// TIA Portal project "hardware_cont" (V17)

(* hardware
DEVICE "S7-1500/ET200MP station_1"  S7-1500 station
   slot 0: "Rail_0"  Rack  6ES7 590-1***0-0AA0
   slot 1: "PLC_1"  CPU 1511-1 PN  6ES7 511-1AK02-0AB0  V2.9
      slot 3: "CPU display_1"  6ES7591-1AA00-0AA0
      slot 32768: "PROFINET interface_1"  X1
         slot 32769: "Port_1"  X1 P1
         slot 32770: "Port_2"  X1 P2
      slot 34817: "Virtual CP interface port_1"  Virtual CP interface port  Virtual CP interface port
   slot 2: "DI 16x24VDC / DQ 16x24VDC/0.5A BA_1"  DI 16x24VDC/DQ 16x24VDC/0.5A BA  6ES7 523-1BL00-0AA0  V1.1
   slot 3: "AI 4xU/I/RTD/TC / AQ 2xU/I ST_1"  AI/AQ 4xU/I/RTD/TC / 2xU/I ST  6ES7 534-7QE00-0AB0  V1.0
   slot 4: "CM PtP RS232 BA_1"  CM PtP RS232 BA  6ES7 540-1AD00-0AA0  V1.0
DEVICE "HMI_2"  TP700 Comfort Outdoor
   slot 0: "HMI_2"  TP700 Comfort Outdoor  6AV2 124-0GC13-0AX0  17.0.0.0
   slot 1: "HMI_RT_2"  TP700 Comfort Outdoor  6AV2 124-0GC13-0AX0  17.0.0.0
   slot 5: "HMI_2.IE_CP_1"  PROFINET Interface  17.0.0.0
      slot 1: "PROFINET Interface_1"  PROFINET Interface
         slot 1: "Port_1"  Port
         slot 2: "Port_2"  Port
   slot 7: "HMI_2.MPI/DP_CP_1"  MPI/DP Interface  17.0.0.0
*)

// ===== PLC "PLC_1"  CPU 1511-1 PN =====

VAR_GLOBAL   // PLC tag table "Default tag table"
   "Open" AT %M0.0 : Bool;
   "Close" AT %M0.1 : Bool;
   "Valve" AT %Q0.0 : Bool;
   "Start" AT %M10.0 : Bool;
   "Stop" AT %M10.1 : Bool;
   "Running" AT %Q0.2 : Bool;
   "Level" AT %MD100 : Real;
   "Val" AT %MD104 : Real;
   "Tank_Level" AT %MD108 : Real;
   "Level2" AT %MD112 : Real;
   "LL_Low" AT %MD116 : Real;
   "Low_LL_Reach" AT %M12.0 : Bool;
   "LL_High" AT %MD120 : Real;
   "High_LL_Reach" AT %M12.2 : Bool;
END_VAR

// folder: System blocks/Program resources

DATA_BLOCK "IEC_Timer_0_DB"   // DB1
{ S7_Optimized_Access := 'TRUE' }
AUTHOR : Simatic
FAMILY : IEC
NAME : IEC_TMR
VERSION : 1.0
// stored: InstanceOfName IEC_TIMER
"IEC_TIMER"
BEGIN
END_DATA_BLOCK

DATA_BLOCK "IEC_Timer_0_DB_1"   // DB2
{ S7_Optimized_Access := 'TRUE' }
AUTHOR : Simatic
FAMILY : IEC
NAME : IEC_TMR
VERSION : 1.0
// stored: InstanceOfName IEC_TIMER
"IEC_TIMER"
BEGIN
END_DATA_BLOCK

// folder: (top level)

ORGANIZATION_BLOCK "Main"   // OB1, LAD, ProgramCycle
TITLE = "Main Program Sweep (Cycle)"
{ S7_Optimized_Access := 'TRUE' }
VERSION : 0.1
   VAR_INPUT
      Initial_Call : Bool;   // Initial call of this OB
      Remanence : Bool;   // =True, if remanent data are available
   END_VAR
BEGIN

REGION Network 1
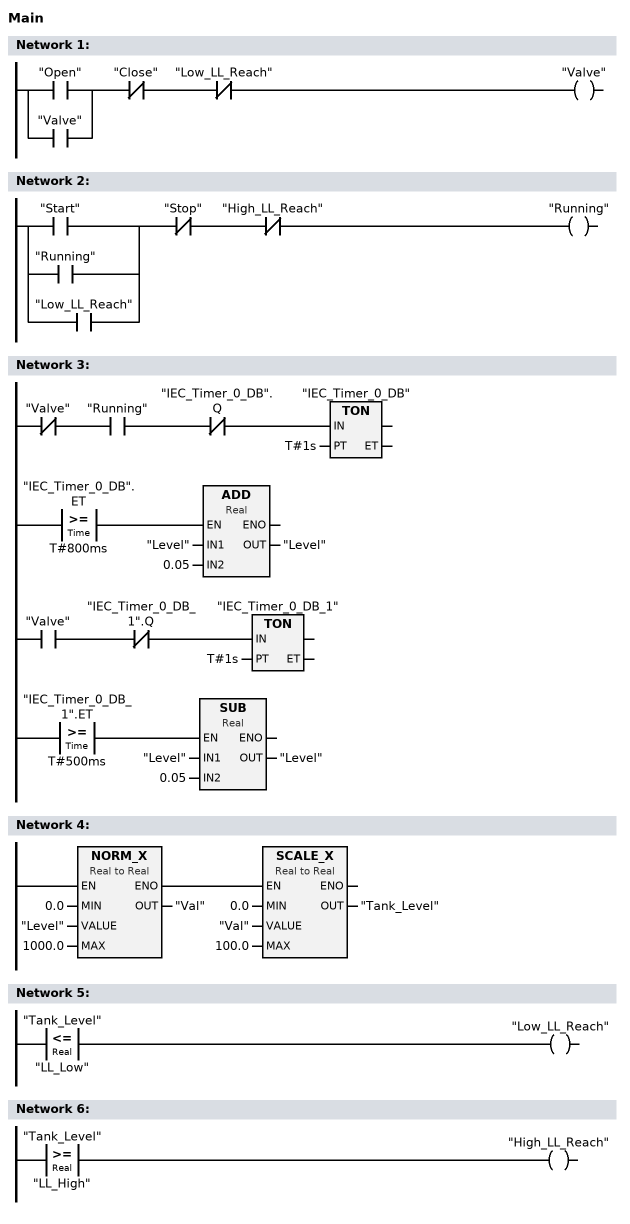
   RUNG wire#powerrail
      Contact( "Open" )
      wire#w1
      I_Contact( "Close" )
      I_Contact( "Low_LL_Reach" )
      Coil( "Valve" )
   END_RUNG
   RUNG wire#powerrail
      Contact( "Valve" )
   END_RUNG wire#w1
   // the same network as SCL:
   "Valve" := ("Open" OR "Valve") AND NOT "Close" AND NOT "Low_LL_Reach";
END_REGION

REGION Network 2
   RUNG wire#powerrail
      Contact( "Start" )
      wire#w1
      I_Contact( "Stop" )
      I_Contact( "High_LL_Reach" )
      Coil( "Running" )
   END_RUNG
   RUNG wire#powerrail
      Contact( "Running" )
   END_RUNG wire#w1
   RUNG wire#powerrail
      Contact( "Low_LL_Reach" )
   END_RUNG wire#w1
   // the same network as SCL:
   "Running" := ("Start" OR "Running" OR "Low_LL_Reach") AND NOT "Stop" AND NOT "High_LL_Reach";
END_REGION

REGION Network 3
   "IEC_Timer_0_DB".TON(IN := NOT "Valve" AND "Running" AND NOT "IEC_Timer_0_DB".Q, PT := T#1s);
   IF "IEC_Timer_0_DB".ET >= T#800ms THEN "Level" := "Level" + 0.05; END_IF;
   "IEC_Timer_0_DB_1".TON(IN := "Valve" AND NOT "IEC_Timer_0_DB_1".Q, PT := T#1s);
   IF "IEC_Timer_0_DB_1".ET >= T#500ms THEN "Level" := "Level" - 0.05; END_IF;
END_REGION

REGION Network 4
   RUNG wire#powerrail
      { S7_Templates := "[SrcType := Real, DestType := Real]" } Normalize(min := 0.0, value := "Level", max := 1000.0, out => "Val")
      { S7_Templates := "[SrcType := Real, DestType := Real]" } Scale(min := 0.0, value := "Val", max := 100.0, out => "Tank_Level")
   END_RUNG
   // the same network as SCL:
   "Val" := NORM_X(MIN := 0.0, VALUE := "Level", MAX := 1000.0);
   "Tank_Level" := SCALE_X(MIN := 0.0, VALUE := "Val", MAX := 100.0);
END_REGION

REGION Network 5
   RUNG wire#powerrail
      { S7_Templates := "SrcType := Real" } LE_Contact(in1 := "Tank_Level", in2 := "LL_Low")
      Coil( "Low_LL_Reach" )
   END_RUNG
   // the same network as SCL:
   "Low_LL_Reach" := "Tank_Level" <= "LL_Low";
END_REGION

REGION Network 6
   RUNG wire#powerrail
      { S7_Templates := "SrcType := Real" } GE_Contact(in1 := "Tank_Level", in2 := "LL_High")
      Coil( "High_LL_Reach" )
   END_RUNG
   // the same network as SCL:
   "High_LL_Reach" := "Tank_Level" >= "LL_High";
END_REGION
END_ORGANIZATION_BLOCK

(* ===== HMI "HMI_RT_2" =====
system functions are stored by id; their names below are inferred from use
connection "HMI_Connection_1": ETHERNET, S7_1500_OMS

HMI tags "Default tag table"
   "Tag_ScreenNumber" : UInt, internal
   "START" : Bool = PLC Open AT %M0.0, 1 s
   "Tank_Level" : Real = PLC Tank_Level AT %MD108, 1 s
   "Start(1)" : Bool = PLC Start AT %M10.0, 1 s
   "Stop" : Bool = PLC Stop AT %M10.1, 1 s
   "Running" : Bool = PLC Running AT %Q0.2, 1 s
   "Close" : Bool = PLC Close AT %M0.1, 1 s
   "Valve" : Bool = PLC Valve AT %Q0.0, 1 s
   "LL_High" : Real = PLC LL_High AT %MD120, 1 s
   "LL_Low" : Real = PLC LL_Low AT %MD116, 1 s

screen "Root screen" 800x420, template "Template_1"
   on GenerateScreen: SetTag("Tag_ScreenNumber", 1)
   TextField "HmiScreenItemData" at 80,166 size 640x25; Text 'Welcome to HMI_2 (TP700 Comfort Outdoor)!'

Template "Template_1" 800x420
   Button "Exit" at 720,360 size 78x58; TextOff 'Exit'; PictureOff "ExitRuntime_TP700_Comfort_Outdoor_TR"; PictureOn "ExitRuntime_TP700_Comfort_Outdoor_TR"
      on Release: StopRuntime(0)
   Button "Template_Button" at 640,360 size 78x58; TextOff 'Text'
   Button "Template_Button_1" at 560,360 size 78x58; TextOff 'Text'
   Button "Template_Button_2" at 480,360 size 78x58; TextOff 'Text'
   Button "Template_Button_3" at 400,360 size 78x58; TextOff 'Text'
   Button "Template_Button_4" at 321,360 size 78x58; TextOff 'Text'
   Button "Template_Button_5" at 241,360 size 78x58; TextOff 'Text'
   Button "Template_Button_6" at 161,360 size 78x58; TextOff 'Text'
   Button "Alarms" at 81,360 size 78x58; TextOff 'Alarms'; PictureOff "AlarmDisplay_TP700_Comfort_Outdoor_TR"; PictureOn "AlarmDisplay_TP700_Comfort_Outdoor_TR"
      on Release: function_ef3f5d25("Alarm window_Unacknowledged", -1)
   Button "Start screen" at 1,360 size 78x58; TextOff 'Start screen'; PictureOff "NavigateHome_TP700_Comfort_Outdoor_TR"; PictureOn "NavigateHome_TP700_Comfort_Outdoor_TR"
      on Release: ActivateScreen("Root screen", 0)

screen "Screen_1" 800x420
   SymbolLibrary "Symbol library_17" at 699,195 size 98x11
      Appearance <- "Valve"
   SymbolLibrary "Symbol library_15" at 270,227 size 13x107
   SymbolLibrary "Symbol library_13" at 154,207 size 111x14
      Appearance <- "Running"
   SymbolLibrary "Symbol library_11" at 581,195 size 135x12
      Appearance <- "Valve"
   SymbolLibrary "Symbol library_9" at 131,54 size 17x167
      Appearance <- "Running"
   SymbolLibrary "Symbol library_7" at 163,21 size 120x19
      Appearance <- "Running"
   SymbolLibrary "Symbol library_6" at 561,40 size 17x48
      Appearance <- "Running"
   SymbolLibrary "Symbol library_5" at 544,21 size 34x36
      Appearance <- "Running"
   SymbolLibrary "Symbol library_4" at 329,21 size 220x19
      Appearance <- "Running"
   SymbolLibrary "Symbol library_1" at 509,78 size 112x183
   SymbolLibrary "Symbol library_2" at 21,177 size 154x78
      Appearance <- "Running"
   SymbolLibrary "Symbol library_3" at 274,5 size 66x39
   SymbolLibrary "Symbol library_8" at 131,21 size 33x36
      Appearance <- "Running"
   SymbolLibrary "Symbol library_10" at 692,152 size 63x60
      Appearance <- "Valve"
   SymbolLibrary "Symbol library_12" at 212,234 size 135x129
   SymbolLibrary "Symbol library_14" at 257,207 size 26x26
      Appearance <- "Running"
   Bar "Bar_1" at 555,91 size 31x105; MinimumValue 0; MaximumValue 100
      ProcessValue <- "Tank_Level"
   SymbolLibrary "Symbol library_16" at 588,71 size 25x50
   Button "Button_1" at 29,328 size 89x21; TextOff 'START'
      on Press: SetBit("Start(1)")
      on Release: ResetBit("Stop")
   Button "Button_2" at 730,94 size 64x17; TextOff 'OPEN'
      on Press: SetBit("START")
      on Release: ResetBit("Close")
   Button "Button_3" at 29,366 size 89x21; TextOff 'STOP'
      on Release: ResetBit("Stop")
      on Press: SetBit("Stop")
   Circle "Circle_1" at 145,339 size 27x27
      Appearance <- "Running"
   IOField "I/O field_1" at 654,305 size 77x32; FormatPattern 999.99
      ProcessValue <- "LL_High"
   IOField "I/O field_2" at 654,355 size 78x32; FormatPattern 999.99
      ProcessValue <- "LL_Low"
   TextField "Text field_1" at 523,312 size 131x23; Text 'SET LEVEL HH'
   TextField "Text field_2" at 523,361 size 131x23; Text 'SET LEVEL LL'
   TextField "Text field_3" at 756,305 size 41x23; Text '(%)'
   TextField "Text field_4" at 756,354 size 41x23; Text '(%)'
   IOField "I/O field_3" at 624,35 size 67x27; FormatPattern 999.99
      ProcessValue <- "Tank_Level"
   TextField "Text field_5" at 600,10 size 120x23; Text 'Level Sensor'
   Button "Button_4" at 729,124 size 65x20; TextOff 'CLOSE'
      on Press: SetBit("Close")
      on Release: ResetBit("Close")
   TextField "Text field_6" at 249,51 size 126x23; Text 'Manual Valve'
   TextField "Text field_7" at 674,212 size 118x23; Text 'Outlet Valve'
   TextField "Text field_8" at 701,40 size 41x23; Text '(%)'
*)